TYPE OperatorStates :
(
	NONE := 0,
	OBSERVER := 1,
	TECH := 2
);
END_TYPE

(* stored: Version 1.1.0.1, ProductVersion 3.1.4019.2
   DUT OperatorStates: Id {d83baffc-c991-4a96-9a1f-02aff60eaaf5} *)
